Fanuc KAREL source: kc00039.KL

-- PROVISIONAL review KL for V770-1; original PC SHA256 9fc92c6d95374bb877f86d91770b16d1e784cdfe3e944a88d4a643aa22e8c7f8
-- Incomplete behavior may be omitted. Consult companion uncertainty JSON. Do not deploy.
PROGRAM KC00039
%NOLOCKGROUP
BEGIN
  -- UNRESOLVED_PC offsets 5-32; opcodes 27,22,22,1C,22,76
  -- UNRESOLVED_PC offsets 37-41; opcodes 7F
END KC00039
